// TIA Portal V19 export
FUNCTION "Analog Scaling" : Void   // FC7, LAD
{ S7_Optimized_Access := 'TRUE' }
// stored: SetENOAutomatically false
BEGIN

REGION Network 1: Line Pressure Scaling
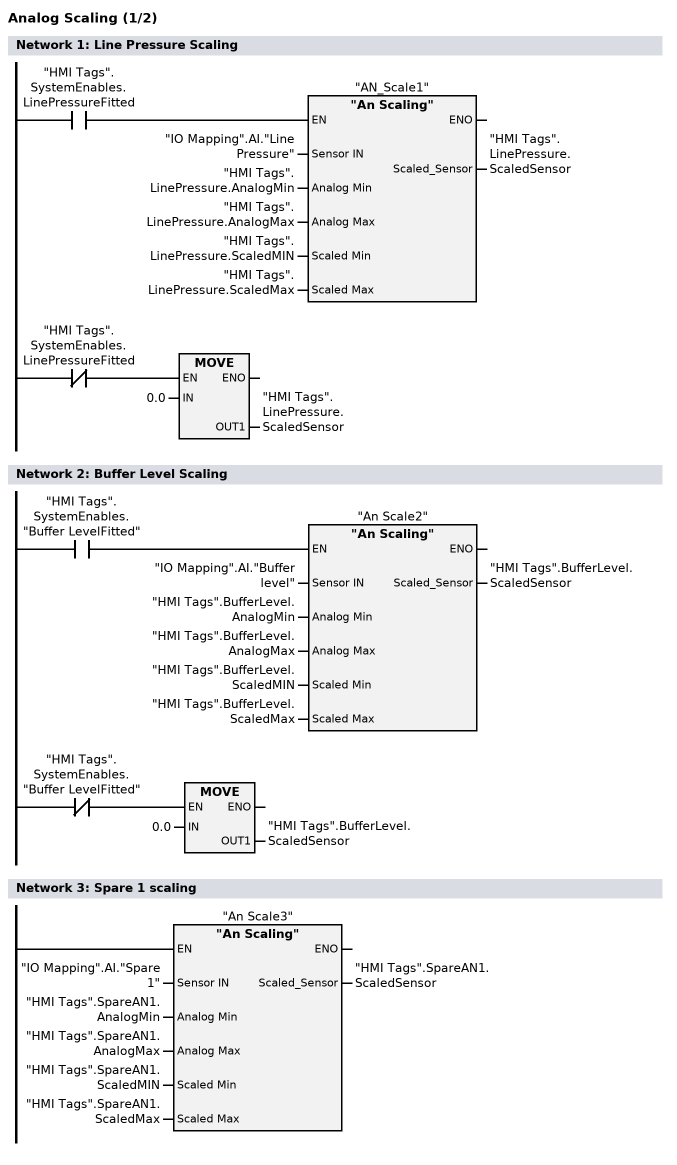
   RUNG wire#powerrail
      Contact( "HMI Tags".SystemEnables.LinePressureFitted )
      "AN_Scale1"("Sensor IN" := "IO Mapping".AI."Line Pressure", "Analog Min" := "HMI Tags".LinePressure.AnalogMin, "Analog Max" := "HMI Tags".LinePressure.AnalogMax, "Scaled Min" := "HMI Tags".LinePressure.ScaledMIN, "Scaled Max" := "HMI Tags".LinePressure.ScaledMax, Scaled_Sensor => "HMI Tags".LinePressure.ScaledSensor)
   END_RUNG
   RUNG wire#powerrail
      I_Contact( "HMI Tags".SystemEnables.LinePressureFitted )
      Move(in := 0.0, out1 => "HMI Tags".LinePressure.ScaledSensor)
   END_RUNG
   // the same network as SCL:
   IF "HMI Tags".SystemEnables.LinePressureFitted THEN
       "AN_Scale1"("Sensor IN" := "IO Mapping".AI."Line Pressure",   // "An Scaling"
                   "Analog Min" := "HMI Tags".LinePressure.AnalogMin,
                   "Analog Max" := "HMI Tags".LinePressure.AnalogMax,
                   "Scaled Min" := "HMI Tags".LinePressure.ScaledMIN,
                   "Scaled Max" := "HMI Tags".LinePressure.ScaledMax,
                   Scaled_Sensor => "HMI Tags".LinePressure.ScaledSensor);
   END_IF;
   IF NOT "HMI Tags".SystemEnables.LinePressureFitted THEN
       "HMI Tags".LinePressure.ScaledSensor := 0.0;
   END_IF;
END_REGION

REGION Network 2: Buffer Level Scaling
   RUNG wire#powerrail
      Contact( "HMI Tags".SystemEnables."Buffer LevelFitted" )
      "An Scale2"("Sensor IN" := "IO Mapping".AI."Buffer level", "Analog Min" := "HMI Tags".BufferLevel.AnalogMin, "Analog Max" := "HMI Tags".BufferLevel.AnalogMax, "Scaled Min" := "HMI Tags".BufferLevel.ScaledMIN, "Scaled Max" := "HMI Tags".BufferLevel.ScaledMax, Scaled_Sensor => "HMI Tags".BufferLevel.ScaledSensor)
   END_RUNG
   RUNG wire#powerrail
      I_Contact( "HMI Tags".SystemEnables."Buffer LevelFitted" )
      Move(in := 0.0, out1 => "HMI Tags".BufferLevel.ScaledSensor)
   END_RUNG
   // the same network as SCL:
   IF "HMI Tags".SystemEnables."Buffer LevelFitted" THEN
       "An Scale2"("Sensor IN" := "IO Mapping".AI."Buffer level",   // "An Scaling"
                   "Analog Min" := "HMI Tags".BufferLevel.AnalogMin,
                   "Analog Max" := "HMI Tags".BufferLevel.AnalogMax,
                   "Scaled Min" := "HMI Tags".BufferLevel.ScaledMIN,
                   "Scaled Max" := "HMI Tags".BufferLevel.ScaledMax,
                   Scaled_Sensor => "HMI Tags".BufferLevel.ScaledSensor);
   END_IF;
   IF NOT "HMI Tags".SystemEnables."Buffer LevelFitted" THEN
       "HMI Tags".BufferLevel.ScaledSensor := 0.0;
   END_IF;
END_REGION

REGION Network 3: Spare 1 scaling
   RUNG wire#powerrail
      "An Scale3"("Sensor IN" := "IO Mapping".AI."Spare 1", "Analog Min" := "HMI Tags".SpareAN1.AnalogMin, "Analog Max" := "HMI Tags".SpareAN1.AnalogMax, "Scaled Min" := "HMI Tags".SpareAN1.ScaledMIN, "Scaled Max" := "HMI Tags".SpareAN1.ScaledMax, Scaled_Sensor => "HMI Tags".SpareAN1.ScaledSensor)
   END_RUNG
   // the same network as SCL:
   "An Scale3"("Sensor IN" := "IO Mapping".AI."Spare 1",   // "An Scaling"
               "Analog Min" := "HMI Tags".SpareAN1.AnalogMin,
               "Analog Max" := "HMI Tags".SpareAN1.AnalogMax,
               "Scaled Min" := "HMI Tags".SpareAN1.ScaledMIN,
               "Scaled Max" := "HMI Tags".SpareAN1.ScaledMax,
               Scaled_Sensor => "HMI Tags".SpareAN1.ScaledSensor);
END_REGION

REGION Network 4: Spare 2 Scaling
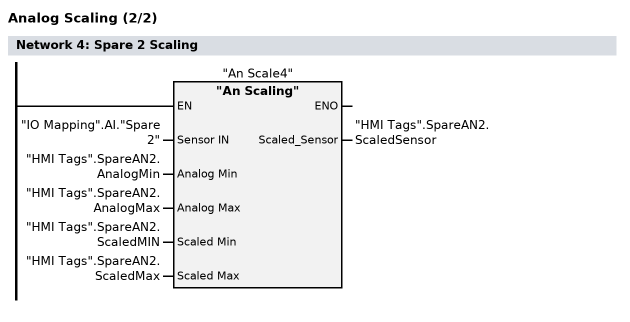
   RUNG wire#powerrail
      "An Scale4"("Sensor IN" := "IO Mapping".AI."Spare 2", "Analog Min" := "HMI Tags".SpareAN2.AnalogMin, "Analog Max" := "HMI Tags".SpareAN2.AnalogMax, "Scaled Min" := "HMI Tags".SpareAN2.ScaledMIN, "Scaled Max" := "HMI Tags".SpareAN2.ScaledMax, Scaled_Sensor => "HMI Tags".SpareAN2.ScaledSensor)
   END_RUNG
   // the same network as SCL:
   "An Scale4"("Sensor IN" := "IO Mapping".AI."Spare 2",   // "An Scaling"
               "Analog Min" := "HMI Tags".SpareAN2.AnalogMin,
               "Analog Max" := "HMI Tags".SpareAN2.AnalogMax,
               "Scaled Min" := "HMI Tags".SpareAN2.ScaledMIN,
               "Scaled Max" := "HMI Tags".SpareAN2.ScaledMax,
               Scaled_Sensor => "HMI Tags".SpareAN2.ScaledSensor);
END_REGION
END_FUNCTION
